{attribute 'pack_mode' := '1'}
    {attribute 'OPC.UA.DA' := '1'}
    {attribute 'OPC.UA.DA.StructuredType' := '1'}
    (*
    ST_RW_Bool_MB_HMI_IgnitionExp
    ==================================================
    Generated from Ignition UDT: RW_Bool_MB
    Total tags: 1
    Generated on: 2025-09-16 12:06:03
    *)
    TYPE ST_RW_Bool_MB_HMI_IgnitionExp :
    STRUCT
        {attribute 'OPC.UA.DA' := '1'}
        {attribute 'OPC.UA.DA.Description' := '{Description}'}
        // {Description}
        Value : BOOL := FALSE;
    END_STRUCT
    END_TYPE

(* stored: Version 1.1.0.1
   DUT ST_RW_Bool_MB_HMI_IgnitionExp: Id {ad785df8-eb2e-4871-845b-8b20b9745cf2} *)
